// TwinCAT 3 PLC project PLC1
// ProgramVersion: 3.1.4024.12
// libraries:
//   Tc2_Standard, * (Beckhoff Automation GmbH)
//   Tc2_System, * (Beckhoff Automation GmbH)
//   Tc3_Module, * (Beckhoff Automation GmbH)
// project tree:
//   FBs/Modules/ FB_LAMP_DIMM.TcPOU, FB_LAMP_ONOFF.TcPOU (not stored)
//   FBs/Room/ FB_ROOM.TcPOU
//   GVLs/ Param.TcGVL (not stored)
//   ITFs/Modules/ I_Lamp.TcIO (not stored)
//   ITFs/Room/ I_Room.TcIO (not stored)
//   / PlcTask.TcTTO (not stored)
//   POUs/ MAIN.TcPOU (not stored)

// ---- FBs/Modules/FB_LAMP_DIMM.TcPOU
{attribute 'reflection'} 
FUNCTION_BLOCK FB_LAMP_DIMM IMPLEMENTS I_Lamp
VAR
	// Hardware control variables
	fOut : REAL;
	fInc : REAL:=0.5;
	iOutHw AT %Q*:INT;
	
	// Instance-path variable
    {attribute 'instance-path'} 
    {attribute 'noinit'} 
    sPath : STRING; 
END_VAR

METHOD OFF : BOOL
// Intensity in 0..100% variable fOut
fOut := fOut - fInc;
IF fOut < 0.0 THEN
	fOut := 0.0;
END_IF

// Conversion to hardware output 0..32767
iOutHw := LIMIT(0,REAL_TO_INT(fOut * 327.67), 32767);
END_METHOD

METHOD ON : BOOL
// Intensity in 0..100% variable fOut
fOut := fOut + fInc;
IF fOut > 100.0 THEN
	fOut := 100.0;
END_IF

// Conversion to hardware output 0..32767
iOutHw := LIMIT(0,REAL_TO_INT(fOut * 327.67), 32767);
END_METHOD

PROPERTY State : STRING
GET
State := CONCAT('Object: ', sPath);
State := CONCAT(State, ' State (%):');
State := CONCAT(State, REAL_TO_STRING(THIS^.fOut));
END_GET
END_PROPERTY

END_FUNCTION_BLOCK

// ---- FBs/Room/FB_ROOM.TcPOU
FUNCTION_BLOCK FB_ROOM IMPLEMENTS I_Room
VAR
	// Array of registered lamps
	iLamps 		: ARRAY[Param.INDEX_START..Param.MAX_LAMPS] OF I_Lamp;
END_VAR

METHOD AddLamp : BOOL
VAR_INPUT
	(* Lamp interface*)
	iLamp	: I_Lamp;
END_VAR

VAR
	// Loop Counter
	nIndex	: INT;
END_VAR
AddLamp := FALSE;
// Check to see if the reference is valid, if not return immediately
IF (iLamp = 0) THEN
	RETURN;
END_IF

// Is the lamp already registered?
FOR nIndex := Param.INDEX_START TO Param.MAX_LAMPS DO
	IF (THIS^.iLamps[nIndex] = iLamp) THEN
		AddLamp := TRUE;
		RETURN;
	END_IF
END_FOR

// Save it to the array if it's not
FOR nIndex := Param.INDEX_START TO  Param.MAX_LAMPS DO
	IF (THIS^.iLamps[nIndex] = 0) THEN
		THIS^.iLamps[nIndex] := iLamp;
		AddLamp := TRUE;
		EXIT;					
	END_IF
END_FOR
END_METHOD

METHOD Control : BOOL
VAR_INPUT
	(* Motion Sensor for the room*)
	bMotionSensor	: BOOL;
END_VAR

VAR
	nIndex: INT;
END_VAR
Control := FALSE;
FOR nIndex := Param.INDEX_START TO  Param.MAX_LAMPS DO
	IF bMotionSensor AND (THIS^.iLamps[nIndex] <> 0) THEN
		iLamps[nIndex].ON();
		Control := TRUE;
	ELSIF (THIS^.iLamps[nIndex] <> 0) THEN
		iLamps[nIndex].OFF();
	END_IF
END_FOR
END_METHOD

METHOD FB_exit : BOOL
VAR_INPUT
	bInCopyCode : BOOL; // if TRUE, the exit method is called for exiting an instance that is copied afterwards (online change).
END_VAR

VAR
	nIndex: INT;
END_VAR
FOR nIndex := 1 TO Param.MAX_LAMPS DO
	iLamps[nIndex] := 16#00;
END_FOR
END_METHOD

METHOD RemoveLamp : BOOL
VAR_INPUT
	(* Lamp interface*)
	iLamp	: I_Lamp;
END_VAR

VAR
	// Loop Counter
	nIndex	: INT;
END_VAR
RemoveLamp := FALSE;

IF (iLamp = 0) THEN
	RETURN;
END_IF

FOR nIndex := Param.INDEX_START TO  Param.MAX_LAMPS DO
	IF (THIS^.iLamps[nIndex] = iLamp) THEN
		THIS^.iLamps[nIndex] := 0;
		RemoveLamp := TRUE;	
	END_IF
END_FOR
END_METHOD

END_FUNCTION_BLOCK
